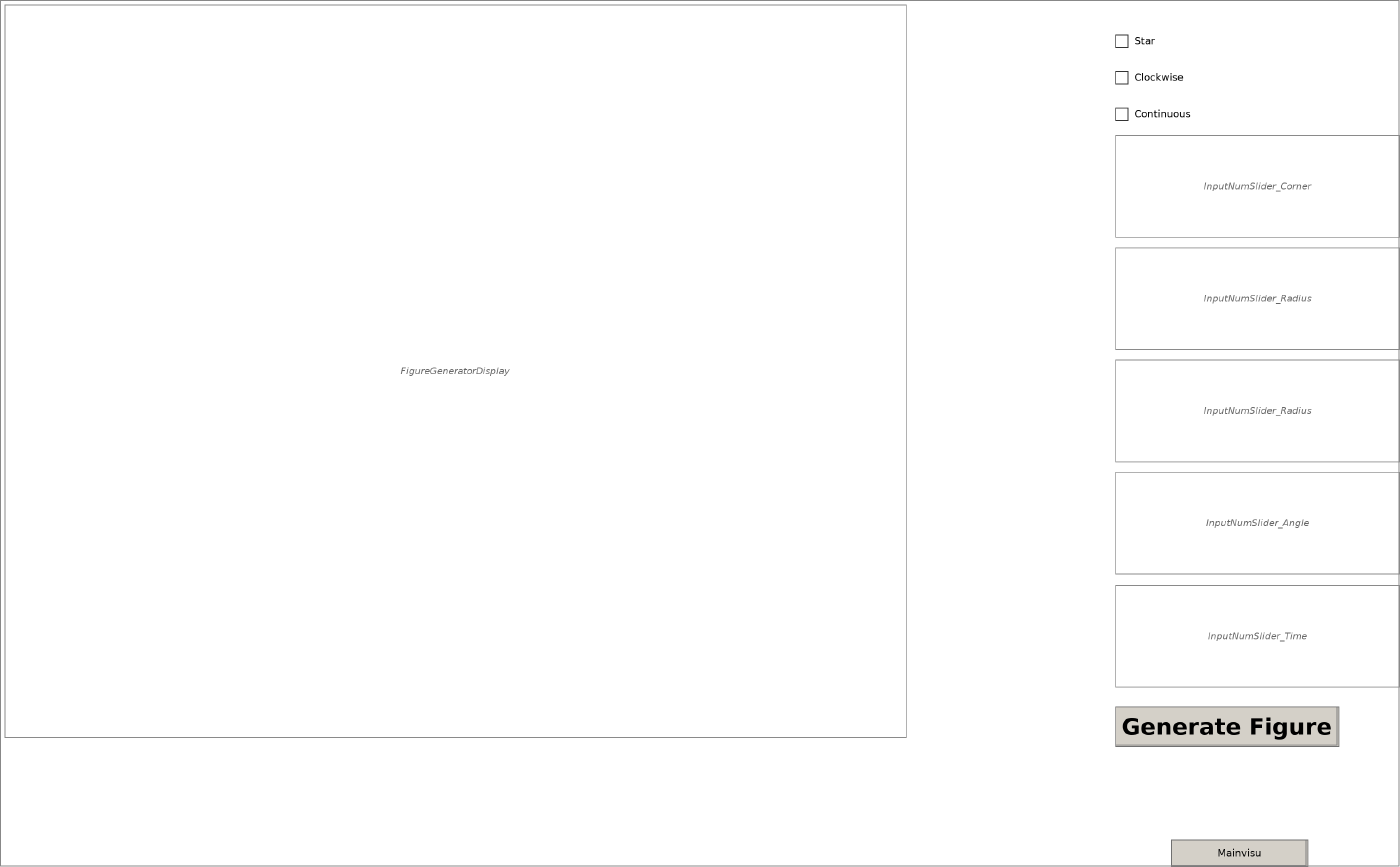
VISUALIZATION FigureGenerator  // 1534x950
    Button (1283,920 150x30), "Mainvisu"
        OnMouseDown: change screen: Mainvisu
    Checkbox (1220,30 150x30), "Star", variable: MAIN.FB_FigureGenerator.bStar
    Checkbox (1220,110 150x30), "Continuous", variable: MAIN.FB_FigureGenerator.bContinus
    Button (1222,774 245x44), "Generate Figure", pressed state: MAIN.FB_FigureGenerator.bGenerate
    Frame (1222,148 312x112)
        shows InputNumSlider_Corner()
    Frame (1222,271 312x112)
        shows InputNumSlider_Radius(number := MAIN.FB_FigureGenerator.rRadius1, name := MAIN.FB_FigureGenerator.sRadius1)
    Frame (1222,394 312x112)
        shows InputNumSlider_Radius(number := MAIN.FB_FigureGenerator.rRadius2, name := MAIN.FB_FigureGenerator.sRadius2)
    Frame (1222,517 312x112)
        shows InputNumSlider_Angle(number := MAIN.FB_FigureGenerator.rAngleOffset)
    Frame (1222,641 312x112)
        shows InputNumSlider_Time(number := MAIN.FB_FigureGenerator.rFigureTime)
    Checkbox (1220,70 150x30), "Clockwise", variable: MAIN.FB_FigureGenerator.bClockwise
    Frame (5,5 988x803)
        shows FigureGeneratorDisplay()
END_VISUALIZATION

(* stored: Version 1.1.0.1, ProductVersion 3.1.4024.12
   Visu FigureGenerator: Id {3d1d9ba4-b19d-452b-a28d-5e0ac4fc0d9a} *)
